# EPICS substitutions: iocBoot/ioc13Saturn1_Linux/roi_to_sca.substitutions
file "$(DXP)/db/roi_to_sca.db"
{
pattern
{P,          M,    D,     N}
{dxpSaturn:, mca1, dxp1:, 0}
{dxpSaturn:, mca1, dxp1:, 1}
{dxpSaturn:, mca1, dxp1:, 2}
{dxpSaturn:, mca1, dxp1:, 3}
{dxpSaturn:, mca1, dxp1:, 4}
{dxpSaturn:, mca1, dxp1:, 5}
{dxpSaturn:, mca1, dxp1:, 6}
{dxpSaturn:, mca1, dxp1:, 7}
{dxpSaturn:, mca1, dxp1:, 8}
{dxpSaturn:, mca1, dxp1:, 9}
{dxpSaturn:, mca1, dxp1:, 10}
{dxpSaturn:, mca1, dxp1:, 11}
{dxpSaturn:, mca1, dxp1:, 12}
{dxpSaturn:, mca1, dxp1:, 13}
{dxpSaturn:, mca1, dxp1:, 14}
{dxpSaturn:, mca1, dxp1:, 15}
}
